DATA_BLOCK "T-84.00"   // DB53
VERSION : 0.1
// stored: AutoNumber false, DBAccessibleFromOPCUA true, DBAccessibleFromWebserver true, InstanceOfName Storage_Tank_Multi_Inload, InstanceOfType FB
"Storage_Tank_Multi_Inload"
BEGIN
END_DATA_BLOCK

DATA_BLOCK "T-85.00"   // DB52
VERSION : 0.1
// stored: AutoNumber false, DBAccessibleFromOPCUA true, DBAccessibleFromWebserver true, InstanceOfName Storage_Tank_Multi_Inload, InstanceOfType FB
"Storage_Tank_Multi_Inload"
BEGIN
END_DATA_BLOCK

DATA_BLOCK "T-02_ChiliAwetan_1"   // DB361
VERSION : 0.1
// stored: AutoNumber false, DBAccessibleFromOPCUA true, DBAccessibleFromWebserver true, InstanceOfName BFT_ChiliAwetan, InstanceOfType FB
"BFT_ChiliAwetan"
BEGIN
END_DATA_BLOCK

DATA_BLOCK "T-03_ChiliAwetan_2"   // DB362
VERSION : 0.1
// stored: AutoNumber false, DBAccessibleFromOPCUA true, DBAccessibleFromWebserver true, InstanceOfName BFT_ChiliAwetan, InstanceOfType FB
"BFT_ChiliAwetan"
BEGIN
END_DATA_BLOCK

DATA_BLOCK "T-04_ChiliAwetan_3"   // DB363
VERSION : 0.1
// stored: AutoNumber false, DBAccessibleFromOPCUA true, DBAccessibleFromWebserver true, InstanceOfName BFT_ChiliAwetan, InstanceOfType FB
"BFT_ChiliAwetan"
BEGIN
END_DATA_BLOCK

DATA_BLOCK "T-05_Tomato"   // DB364
VERSION : 0.1
// stored: AutoNumber false, DBAccessibleFromOPCUA true, DBAccessibleFromWebserver true, InstanceOfName BFT_Tomato, InstanceOfType FB
"BFT_Tomato"
BEGIN
END_DATA_BLOCK

DATA_BLOCK "T-06_ChiliFresh_1"   // DB365
VERSION : 0.1
// stored: AutoNumber false, DBAccessibleFromOPCUA true, DBAccessibleFromWebserver true, InstanceOfName BFT_ChiliFresh, InstanceOfType FB
"BFT_ChiliFresh"
BEGIN
END_DATA_BLOCK

DATA_BLOCK "T-07_ChiliFresh_2"   // DB366
VERSION : 0.1
// stored: AutoNumber false, DBAccessibleFromOPCUA true, DBAccessibleFromWebserver true, InstanceOfName BFT_ChiliFresh, InstanceOfType FB
"BFT_ChiliFresh"
BEGIN
END_DATA_BLOCK

DATA_BLOCK "T-08_ChiliFresh_3"   // DB367
VERSION : 0.1
// stored: AutoNumber false, DBAccessibleFromOPCUA true, DBAccessibleFromWebserver true, InstanceOfName BFT_ChiliFresh, InstanceOfType FB
"BFT_ChiliFresh"
BEGIN
END_DATA_BLOCK

DATA_BLOCK "T-09_Garlic"   // DB368
VERSION : 0.1
// stored: AutoNumber false, DBAccessibleFromOPCUA true, DBAccessibleFromWebserver true, InstanceOfName BFT_Garlic, InstanceOfType FB
"BFT_Garlic"
BEGIN
END_DATA_BLOCK

DATA_BLOCK "T-10_Vinegar"   // DB369
VERSION : 0.1
// stored: AutoNumber false, DBAccessibleFromOPCUA true, DBAccessibleFromWebserver true, InstanceOfName BFT_Vinegar, InstanceOfType FB
"BFT_Vinegar"
BEGIN
END_DATA_BLOCK

DATA_BLOCK "T-51_HW"   // DB370
VERSION : 0.1
// stored: AutoNumber false, DBAccessibleFromOPCUA true, DBAccessibleFromWebserver true, InstanceOfName Hot_Water, InstanceOfType FB
"Hot_Water"
BEGIN
END_DATA_BLOCK

DATA_BLOCK "BFT-61"   // DB111
VERSION : 0.1
// stored: AutoNumber false, DBAccessibleFromOPCUA true, DBAccessibleFromWebserver true, InstanceOfName Buffer_Tank, InstanceOfType FB
"Buffer_Tank"
BEGIN
END_DATA_BLOCK

DATA_BLOCK "BFT-64"   // DB112
VERSION : 0.1
// stored: AutoNumber false, DBAccessibleFromOPCUA true, DBAccessibleFromWebserver true, InstanceOfName Buffer_Tank, InstanceOfType FB
"Buffer_Tank"
BEGIN
END_DATA_BLOCK

DATA_BLOCK "BFT-65"   // DB113
VERSION : 0.1
// stored: AutoNumber false, DBAccessibleFromOPCUA true, DBAccessibleFromWebserver true, InstanceOfName Buffer_Tank, InstanceOfType FB
"Buffer_Tank"
BEGIN
END_DATA_BLOCK

DATA_BLOCK "BFT-66"   // DB114
VERSION : 0.1
// stored: AutoNumber false, DBAccessibleFromOPCUA true, DBAccessibleFromWebserver true, InstanceOfName Buffer_Tank, InstanceOfType FB
"Buffer_Tank"
BEGIN
END_DATA_BLOCK

DATA_BLOCK "BFT-67"   // DB115
VERSION : 0.1
// stored: AutoNumber false, DBAccessibleFromOPCUA true, DBAccessibleFromWebserver true, InstanceOfName Buffer_Tank, InstanceOfType FB
"Buffer_Tank"
BEGIN
END_DATA_BLOCK

DATA_BLOCK "BFT-68"   // DB116
VERSION : 0.1
// stored: AutoNumber false, DBAccessibleFromOPCUA true, DBAccessibleFromWebserver true, InstanceOfName Buffer_Tank, InstanceOfType FB
"Buffer_Tank"
BEGIN
END_DATA_BLOCK

DATA_BLOCK "Danfos_VSD_DB"   // DB46
VERSION : 0.1
// stored: AutoNumber false, DBAccessibleFromOPCUA true, DBAccessibleFromWebserver true, InstanceOfName Danfos_VSD, InstanceOfType FB
"Danfos_VSD"
BEGIN
END_DATA_BLOCK

DATA_BLOCK "IO Motor MCC Panel Blending_DB"   // DB5
VERSION : 0.1
// stored: AutoNumber true, DBAccessibleFromOPCUA true, DBAccessibleFromWebserver true, InstanceOfName IO Motor MCC Panel Blending, InstanceOfType FB
"IO Motor MCC Panel Blending"
BEGIN
   "XA-20.00".IN_SP_Speed := 5.0;
   "XA-21.00".IN_SP_Speed := 5.0;
   "P-21.01".IN_SP_Speed := 5.0;
   "XA-30.00".IN_SP_Speed := 5.0;
   "XA-31.00".IN_SP_Speed := 5.0;
   "P-31.01".IN_SP_Speed := 5.0;
   "P-32.01".IN_SP_Speed := 5.0;
   "P-32.03".IN_SP_Speed := 5.0;
END_DATA_BLOCK

DATA_BLOCK "P21.01Dan"   // DB23
VERSION : 0.1
// stored: AutoNumber true, DBAccessibleFromOPCUA true, DBAccessibleFromWebserver true, InstanceOfName Danfos_VSD, InstanceOfType FB
"Danfos_VSD"
BEGIN
END_DATA_BLOCK

DATA_BLOCK "P22.01Dan"   // DB22
VERSION : 0.1
// stored: AutoNumber true, DBAccessibleFromOPCUA true, DBAccessibleFromWebserver true, InstanceOfName Danfos_VSD, InstanceOfType FB
"Danfos_VSD"
BEGIN
END_DATA_BLOCK

DATA_BLOCK "IO Analog Homomixer_DB"   // DB2
VERSION : 0.1
// stored: AutoNumber true, DBAccessibleFromOPCUA true, DBAccessibleFromWebserver true, InstanceOfName IO Analog Homomixer, InstanceOfType FB
"IO Analog Homomixer"
BEGIN
END_DATA_BLOCK

DATA_BLOCK "IO Digital Homomixer_DB"   // DB3
VERSION : 0.1
// stored: AutoNumber true, DBAccessibleFromOPCUA true, DBAccessibleFromWebserver true, InstanceOfName IO Digital Homomixer, InstanceOfType FB
"IO Digital Homomixer"
BEGIN
END_DATA_BLOCK

DATA_BLOCK "IO Valve Homomixer_DB"   // DB4
VERSION : 0.1
// stored: AutoNumber true, DBAccessibleFromOPCUA true, DBAccessibleFromWebserver true, InstanceOfName IO Valve Homomixer, InstanceOfType FB
"IO Valve Homomixer"
BEGIN
END_DATA_BLOCK

DATA_BLOCK "IO Analog Blending_DB"   // DB6
VERSION : 0.1
// stored: AutoNumber true, DBAccessibleFromOPCUA true, DBAccessibleFromWebserver true, InstanceOfName IO Analog Blending, InstanceOfType FB
"IO Analog Blending"
BEGIN
END_DATA_BLOCK

DATA_BLOCK "IO Digital Blending_DB"   // DB7
VERSION : 0.1
// stored: AutoNumber true, DBAccessibleFromOPCUA true, DBAccessibleFromWebserver true, InstanceOfName IO Digital Blending, InstanceOfType FB
"IO Digital Blending"
BEGIN
END_DATA_BLOCK

DATA_BLOCK "IO_Valve_Blend20_DB"   // DB28
VERSION : 0.1
// stored: AutoNumber true, DBAccessibleFromOPCUA true, DBAccessibleFromWebserver true, InstanceOfName IO_Valve_Blend20, InstanceOfType FB
"IO_Valve_Blend20"
BEGIN
END_DATA_BLOCK

DATA_BLOCK "IO_Valve_Blend21_DB"   // DB39
VERSION : 0.1
// stored: AutoNumber true, DBAccessibleFromOPCUA true, DBAccessibleFromWebserver true, InstanceOfName IO_Valve_Blend21, InstanceOfType FB
"IO_Valve_Blend21"
BEGIN
END_DATA_BLOCK

DATA_BLOCK "IO_Valve_Blend30_DB"   // DB60
VERSION : 0.1
// stored: AutoNumber true, DBAccessibleFromOPCUA true, DBAccessibleFromWebserver true, InstanceOfName IO_Valve_Blend30, InstanceOfType FB
"IO_Valve_Blend30"
BEGIN
END_DATA_BLOCK

DATA_BLOCK "IO_Valve_Blend31_DB"   // DB61
VERSION : 0.1
// stored: AutoNumber true, DBAccessibleFromOPCUA true, DBAccessibleFromWebserver true, InstanceOfName IO_Valve_Blend31, InstanceOfType FB
"IO_Valve_Blend31"
BEGIN
END_DATA_BLOCK

DATA_BLOCK "IO_Valve_Blend40_DB"   // DB26
VERSION : 0.1
// stored: AutoNumber true, DBAccessibleFromOPCUA true, DBAccessibleFromWebserver true, InstanceOfName IO_Valve_Blend40, InstanceOfType FB
"IO_Valve_Blend40"
BEGIN
END_DATA_BLOCK

DATA_BLOCK "IO_Valve_Blend41_DB"   // DB62
VERSION : 0.1
// stored: AutoNumber true, DBAccessibleFromOPCUA true, DBAccessibleFromWebserver true, InstanceOfName IO_Valve_Blend41, InstanceOfType FB
"IO_Valve_Blend41"
BEGIN
END_DATA_BLOCK

DATA_BLOCK "IO_Valve_Blending_DB"   // DB8
VERSION : 0.1
// stored: AutoNumber true, DBAccessibleFromOPCUA true, DBAccessibleFromWebserver true, InstanceOfName IO_Valve_Blending, InstanceOfType FB
"IO_Valve_Blending"
BEGIN
   "AV-20.02".OPdwCmd := 16#0008_0000;
   "AV-20.03".OPdwCmd := 16#0008_0000;
   "AV-20.04".OPdwCmd := 16#0008_0000;
   "AV-20.05".OPdwCmd := 16#0008_0000;
   "AV-20.06".OPdwCmd := 16#0008_0000;
   "AV-20.07".OPdwCmd := 16#0008_0000;
   "AV-20.08".OPdwCmd := 16#0008_0000;
   "AV-20.09".OPdwCmd := 16#0008_0000;
   "AV-20.10".OPdwCmd := 16#0008_0000;
   "AV-20.11".OPdwCmd := 16#0008_0000;
   "AV-20.12".OPdwCmd := 16#0008_0000;
   "AV-20.13".OPdwCmd := 16#0008_0000;
   "AV-20.14".OPdwCmd := 16#0008_0000;
   "AV-20.15".OPdwCmd := 16#0008_0000;
   "AV-20.16".OPdwCmd := 16#0008_0000;
   "AV-20.17".OPdwCmd := 16#0008_0000;
   "AV-20.31".OPdwCmd := 16#0008_0000;
   "AV-20.32".OPdwCmd := 16#0008_0000;
   "AV-20.33".OPdwCmd := 16#0008_0000;
   "AV-20.34".OPdwCmd := 16#0008_0000;
   "AV-20.35".OPdwCmd := 16#0008_0000;
   "AV-20.36".OPdwCmd := 16#0008_0000;
   "AV-20.37".OPdwCmd := 16#0008_0000;
   "AV-20.38".OPdwCmd := 16#0008_0000;
   "AV-20.39".OPdwCmd := 16#0008_0000;
   "AV-20.40".OPdwCmd := 16#0008_0000;
   "AV-20.41".OPdwCmd := 16#0008_0000;
   "AV-21.01".OPdwCmd := 16#0008_0000;
   "AV-21.02".OPdwCmd := 16#0008_0000;
   "AV-21.03".OPdwCmd := 16#0008_0000;
   "AV-21.04".OPdwCmd := 16#0008_0000;
   "AV-21.05".OPdwCmd := 16#0008_0000;
   "AV-21.06".OPdwCmd := 16#0008_0000;
   "AV-21.07".OPdwCmd := 16#0008_0000;
   "AV-21.08".OPdwCmd := 16#0008_0000;
   "AV-21.09".OPdwCmd := 16#0008_0000;
   "AV-21.10".OPdwCmd := 16#0008_0000;
   "AV-21.11".OPdwCmd := 16#0008_0000;
   "AV-21.12".OPdwCmd := 16#0008_0000;
   "AV-21.13".OPdwCmd := 16#0008_0000;
   "AV-21.14".OPdwCmd := 16#0008_0000;
   "AV-21.15".OPdwCmd := 16#0008_0000;
   "AV-21.16".OPdwCmd := 16#0008_0000;
   "AV-21.17".OPdwCmd := 16#0008_0000;
   "AV-21.18".OPdwCmd := 16#0008_0000;
   "AV-21.31".OPdwCmd := 16#0008_0000;
   "AV-21.32".OPdwCmd := 16#0008_0000;
   "AV-21.33".OPdwCmd := 16#0008_0000;
   "AV-21.34".OPdwCmd := 16#0008_0000;
   "AV-21.35".OPdwCmd := 16#0008_0000;
   "AV-21.36".OPdwCmd := 16#0008_0000;
   "AV-21.37".OPdwCmd := 16#0008_0000;
   "AV-21.38".OPdwCmd := 16#0008_0000;
   "AV-21.39".OPdwCmd := 16#0008_0000;
   "AV-21.40".OPdwCmd := 16#0008_0000;
   "AV-21.41".OPdwCmd := 16#0008_0000;
   "AV-22.01".OPdwCmd := 16#0008_0000;
   "AV-22.02".OPdwCmd := 16#0008_0000;
   "AV-22.03".OPdwCmd := 16#0008_0000;
   "AV-22.06".OPdwCmd := 16#0008_0000;
   "AV-22.11".OPdwCmd := 16#0008_0000;
   "AV-22.21".OPdwCmd := 16#0008_0000;
   "AV-22.22".OPdwCmd := 16#0008_0000;
   "AV-30.01".OPdwCmd := 16#0008_0000;
   "AV-30.02".OPdwCmd := 16#0008_0000;
   "AV-30.03".OPdwCmd := 16#0008_0000;
   "AV-30.04".OPdwCmd := 16#0008_0000;
   "AV-30.05".OPdwCmd := 16#0008_0000;
   "AV-30.06".OPdwCmd := 16#0008_0000;
   "AV-30.07".OPdwCmd := 16#0008_0000;
   "AV-30.08".OPdwCmd := 16#0008_0000;
   "AV-30.09".OPdwCmd := 16#0008_0000;
   "AV-30.10".OPdwCmd := 16#0008_0000;
   "AV-30.11".OPdwCmd := 16#0008_0000;
   "AV-30.12".OPdwCmd := 16#0008_0000;
   "AV-30.13".OPdwCmd := 16#0008_0000;
   "AV-30.14".OPdwCmd := 16#0008_0000;
   "AV-30.15".OPdwCmd := 16#0008_0000;
   "AV-30.16".OPdwCmd := 16#0008_0000;
   "AV-30.17".OPdwCmd := 16#0008_0000;
   "AV-30.31".OPdwCmd := 16#0008_0000;
   "AV-30.32".OPdwCmd := 16#0008_0000;
   "AV-30.33".OPdwCmd := 16#0008_0000;
   "AV-30.34".OPdwCmd := 16#0008_0000;
   "AV-30.35".OPdwCmd := 16#0008_0000;
   "AV-30.36".OPdwCmd := 16#0008_0000;
   "AV-30.37".OPdwCmd := 16#0008_0000;
   "AV-30.38".OPdwCmd := 16#0008_0000;
   "AV-30.39".OPdwCmd := 16#0008_0000;
   "AV-30.40".OPdwCmd := 16#0008_0000;
   "AV-30.41".OPdwCmd := 16#0008_0000;
   "AV-31.01".OPdwCmd := 16#0008_0000;
   "AV-31.02".OPdwCmd := 16#0008_0000;
   "AV-31.03".OPdwCmd := 16#0008_0000;
   "AV-31.04".OPdwCmd := 16#0008_0000;
   "AV-31.05".OPdwCmd := 16#0008_0000;
   "AV-31.06".OPdwCmd := 16#0008_0000;
   "AV-31.07".OPdwCmd := 16#0008_0000;
   "AV-31.08".OPdwCmd := 16#0008_0000;
   "AV-31.09".OPdwCmd := 16#0008_0000;
   "AV-31.10".OPdwCmd := 16#0008_0000;
   "AV-31.11".OPdwCmd := 16#0008_0000;
   "AV-31.12".OPdwCmd := 16#0008_0000;
   "AV-31.13".OPdwCmd := 16#0008_0000;
   "AV-31.14".OPdwCmd := 16#0008_0000;
   "AV-31.15".OPdwCmd := 16#0008_0000;
   "AV-31.16".OPdwCmd := 16#0008_0000;
   "AV-31.17".OPdwCmd := 16#0008_0000;
   "AV-31.18".OPdwCmd := 16#0008_0000;
   "AV-31.31".OPdwCmd := 16#0008_0000;
   "AV-31.32".OPdwCmd := 16#0008_0000;
   "AV-31.33".OPdwCmd := 16#0008_0000;
   "AV-31.34".OPdwCmd := 16#0008_0000;
   "AV-31.35".OPdwCmd := 16#0008_0000;
   "AV-31.36".OPdwCmd := 16#0008_0000;
   "AV-31.37".OPdwCmd := 16#0008_0000;
   "AV-31.38".OPdwCmd := 16#0008_0000;
   "AV-31.39".OPdwCmd := 16#0008_0000;
   "AV-31.40".OPdwCmd := 16#0008_0000;
   "AV-31.41".OPdwCmd := 16#0008_0000;
   "AV-31.51".OPdwCmd := 16#0008_0000;
   "AV-31.52".OPdwCmd := 16#0008_0000;
   "AV-31.53".OPdwCmd := 16#0008_0000;
   "AV-31.54".OPdwCmd := 16#0008_0000;
   "AV-31.55".OPdwCmd := 16#0008_0000;
   "AV-31.56".OPdwCmd := 16#0008_0000;
   "AV-31.57".OPdwCmd := 16#0008_0000;
   "AV-31.58".OPdwCmd := 16#0008_0000;
   "AV-31.59".OPdwCmd := 16#0008_0000;
   "AV-31.60".OPdwCmd := 16#0008_0000;
   "AV-31.61".OPdwCmd := 16#0008_0000;
   "AV-31.62".OPdwCmd := 16#0008_0000;
   "AV-32.01".OPdwCmd := 16#0008_0000;
   "AV-32.02".OPdwCmd := 16#0008_0000;
   "AV-32.03".OPdwCmd := 16#0008_0000;
   "AV-32.06".OPdwCmd := 16#0008_0000;
   "AV-32.11".OPdwCmd := 16#0008_0000;
   "AV-32.21".OPdwCmd := 16#0008_0000;
   "AV-32.22".OPdwCmd := 16#0008_0000;
   "AV-20.42".OPdwCmd := 16#0008_0000;
   "AV-21.42".OPdwCmd := 16#0008_0000;
   "AV-22.04".OPdwCmd := 16#0008_0000;
   "AV-22.05".OPdwCmd := 16#0008_0000;
   "AV-30.42".OPdwCmd := 16#0008_0000;
   "AV-31.42".OPdwCmd := 16#0008_0000;
   "AV-32.04".OPdwCmd := 16#0008_0000;
   "AV-32.05".OPdwCmd := 16#0008_0000;
END_DATA_BLOCK

DATA_BLOCK "IO Analog Storage_DB"   // DB9
VERSION : 0.1
// stored: AutoNumber true, DBAccessibleFromOPCUA true, DBAccessibleFromWebserver true, InstanceOfName IO Analog Storage, InstanceOfType FB
"IO Analog Storage"
BEGIN
END_DATA_BLOCK

DATA_BLOCK "IO_Digital_Storage_DB"   // DB44
VERSION : 0.1
// stored: AutoNumber true, DBAccessibleFromOPCUA true, DBAccessibleFromWebserver true, InstanceOfName IO_Digital_Storage, InstanceOfType FB
"IO_Digital_Storage"
BEGIN
END_DATA_BLOCK

DATA_BLOCK "IO_Valve_Storage_DB"   // DB11
VERSION : 0.1
// stored: AutoNumber true, DBAccessibleFromOPCUA true, DBAccessibleFromWebserver true, InstanceOfName IO_Valve_Storage, InstanceOfType FB
"IO_Valve_Storage"
BEGIN
END_DATA_BLOCK

DATA_BLOCK "IO Motor MCC Preparation_DB"   // DB12
VERSION : 0.1
// stored: AutoNumber true, DBAccessibleFromOPCUA true, DBAccessibleFromWebserver true, InstanceOfName IO Motor MCC Preparation, InstanceOfType FB
"IO Motor MCC Preparation"
BEGIN
END_DATA_BLOCK

DATA_BLOCK "IO Analog Preparation_DB"   // DB13
VERSION : 0.1
// stored: AutoNumber true, DBAccessibleFromOPCUA true, DBAccessibleFromWebserver true, InstanceOfName IO Analog Preparation, InstanceOfType FB
"IO Analog Preparation"
BEGIN
END_DATA_BLOCK

DATA_BLOCK "IO Digital Preparation_DB"   // DB14
VERSION : 0.1
// stored: AutoNumber true, DBAccessibleFromOPCUA true, DBAccessibleFromWebserver true, InstanceOfName IO Digital Preparation, InstanceOfType FB
"IO Digital Preparation"
BEGIN
END_DATA_BLOCK

DATA_BLOCK "IO_Valve_T01_HWT"   // DB301
VERSION : 0.1
// stored: AutoNumber false, DBAccessibleFromOPCUA true, DBAccessibleFromWebserver true, InstanceOfName IO Valve T01 HWT, InstanceOfType FB
"IO Valve T01 HWT"
BEGIN
END_DATA_BLOCK

DATA_BLOCK "IO_Valve_T02_Chili"   // DB302
VERSION : 0.1
// stored: AutoNumber false, DBAccessibleFromOPCUA true, DBAccessibleFromWebserver true, InstanceOfName IO Valve T02 Chili, InstanceOfType FB
"IO Valve T02 Chili"
BEGIN
END_DATA_BLOCK

DATA_BLOCK "IO_Valve_T03_Chili"   // DB303
VERSION : 0.1
// stored: AutoNumber false, DBAccessibleFromOPCUA true, DBAccessibleFromWebserver true, InstanceOfName IO Valve T03 Chili, InstanceOfType FB
"IO Valve T03 Chili"
BEGIN
END_DATA_BLOCK

DATA_BLOCK "IO_Valve_T04_Chili"   // DB304
VERSION : 0.1
// stored: AutoNumber false, DBAccessibleFromOPCUA true, DBAccessibleFromWebserver true, InstanceOfName IO Valve T04 Chili, InstanceOfType FB
"IO Valve T04 Chili"
BEGIN
END_DATA_BLOCK

DATA_BLOCK "IO_Valve_T05_Tomato"   // DB305
VERSION : 0.1
// stored: AutoNumber false, DBAccessibleFromOPCUA true, DBAccessibleFromWebserver true, InstanceOfName IO Valve T05 Tomato, InstanceOfType FB
"IO Valve T05 Tomato"
BEGIN
END_DATA_BLOCK

DATA_BLOCK "IO_Valve_T06_FreshChili"   // DB306
VERSION : 0.1
// stored: AutoNumber false, DBAccessibleFromOPCUA true, DBAccessibleFromWebserver true, InstanceOfName IO Valve T06 FreshChili, InstanceOfType FB
"IO Valve T06 FreshChili"
BEGIN
END_DATA_BLOCK

DATA_BLOCK "IO_Valve_T07_FreshChili"   // DB307
VERSION : 0.1
// stored: AutoNumber false, DBAccessibleFromOPCUA true, DBAccessibleFromWebserver true, InstanceOfName IO Valve T07 FreshChili, InstanceOfType FB
"IO Valve T07 FreshChili"
BEGIN
END_DATA_BLOCK

DATA_BLOCK "IO_Valve_T08_FreshChili"   // DB308
VERSION : 0.1
// stored: AutoNumber false, DBAccessibleFromOPCUA true, DBAccessibleFromWebserver true, InstanceOfName IO Valve T08 FreshChili, InstanceOfType FB
"IO Valve T08 FreshChili"
BEGIN
END_DATA_BLOCK

DATA_BLOCK "IO_Valve_T09_Garlic"   // DB309
VERSION : 0.1
// stored: AutoNumber false, DBAccessibleFromOPCUA true, DBAccessibleFromWebserver true, InstanceOfName IO Valve T09 Garlic, InstanceOfType FB
"IO Valve T09 Garlic"
BEGIN
END_DATA_BLOCK

DATA_BLOCK "IO_Valve_T10_Vinegar"   // DB310
VERSION : 0.1
// stored: AutoNumber false, DBAccessibleFromOPCUA true, DBAccessibleFromWebserver true, InstanceOfName IO Valve T10 Vinegar, InstanceOfType FB
"IO Valve T10 Vinegar"
BEGIN
END_DATA_BLOCK

DATA_BLOCK "IO_Valve_T51_HW"   // DB311
VERSION : 0.1
// stored: AutoNumber false, DBAccessibleFromOPCUA true, DBAccessibleFromWebserver true, InstanceOfName IO Valve T51 HotWaterLine, InstanceOfType FB
"IO Valve T51 HotWaterLine"
BEGIN
END_DATA_BLOCK

DATA_BLOCK "IO_Valve_Buffer_DB"   // DB64
VERSION : 0.1
// stored: AutoNumber true, DBAccessibleFromOPCUA true, DBAccessibleFromWebserver true, InstanceOfName IO_Valve_Buffer, InstanceOfType FB
"IO_Valve_Buffer"
BEGIN
END_DATA_BLOCK

DATA_BLOCK "Totalizer_FT-00.01"   // DB381
VERSION : 0.1
// stored: AutoNumber false, DBAccessibleFromOPCUA true, DBAccessibleFromWebserver true, InstanceOfName Totalizer, InstanceOfType FB
"Totalizer"
BEGIN
END_DATA_BLOCK

DATA_BLOCK "Totalizer_FT-02.01"   // DB382
VERSION : 0.1
// stored: AutoNumber false, DBAccessibleFromOPCUA true, DBAccessibleFromWebserver true, InstanceOfName Totalizer, InstanceOfType FB
"Totalizer"
BEGIN
END_DATA_BLOCK

DATA_BLOCK "Totalizer_FT-03.01"   // DB383
VERSION : 0.1
// stored: AutoNumber false, DBAccessibleFromOPCUA true, DBAccessibleFromWebserver true, InstanceOfName Totalizer, InstanceOfType FB
"Totalizer"
BEGIN
END_DATA_BLOCK

DATA_BLOCK "Totalizer_FT-04.01"   // DB384
VERSION : 0.1
// stored: AutoNumber false, DBAccessibleFromOPCUA true, DBAccessibleFromWebserver true, InstanceOfName Totalizer, InstanceOfType FB
"Totalizer"
BEGIN
END_DATA_BLOCK

DATA_BLOCK "Totalizer_FT-05.01"   // DB385
VERSION : 0.1
// stored: AutoNumber false, DBAccessibleFromOPCUA true, DBAccessibleFromWebserver true, InstanceOfName Totalizer, InstanceOfType FB
"Totalizer"
BEGIN
END_DATA_BLOCK

DATA_BLOCK "Totalizer_FT-06.01"   // DB386
VERSION : 0.1
// stored: AutoNumber false, DBAccessibleFromOPCUA true, DBAccessibleFromWebserver true, InstanceOfName Totalizer, InstanceOfType FB
"Totalizer"
BEGIN
END_DATA_BLOCK

DATA_BLOCK "Totalizer_FT-07.01"   // DB387
VERSION : 0.1
// stored: AutoNumber false, DBAccessibleFromOPCUA true, DBAccessibleFromWebserver true, InstanceOfName Totalizer, InstanceOfType FB
"Totalizer"
BEGIN
END_DATA_BLOCK

DATA_BLOCK "Totalizer_FT-08.01"   // DB388
VERSION : 0.1
// stored: AutoNumber false, DBAccessibleFromOPCUA true, DBAccessibleFromWebserver true, InstanceOfName Totalizer, InstanceOfType FB
"Totalizer"
BEGIN
END_DATA_BLOCK

DATA_BLOCK "Totalizer_FT-09.01"   // DB389
VERSION : 0.1
// stored: AutoNumber false, DBAccessibleFromOPCUA true, DBAccessibleFromWebserver true, InstanceOfName Totalizer, InstanceOfType FB
"Totalizer"
BEGIN
END_DATA_BLOCK

DATA_BLOCK "Totalizer_FT-10.01"   // DB390
VERSION : 0.1
// stored: AutoNumber false, DBAccessibleFromOPCUA true, DBAccessibleFromWebserver true, InstanceOfName Totalizer, InstanceOfType FB
"Totalizer"
BEGIN
END_DATA_BLOCK

DATA_BLOCK "Totalizer_FT-12.01"   // DB393
VERSION : 0.1
// stored: AutoNumber false, DBAccessibleFromOPCUA true, DBAccessibleFromWebserver true, InstanceOfName Totalizer, InstanceOfType FB
"Totalizer"
BEGIN
END_DATA_BLOCK

DATA_BLOCK "Totalizer_FT-12.02"   // DB394
VERSION : 0.1
// stored: AutoNumber false, DBAccessibleFromOPCUA true, DBAccessibleFromWebserver true, InstanceOfName Totalizer, InstanceOfType FB
"Totalizer"
BEGIN
END_DATA_BLOCK

DATA_BLOCK "Totalizer_FT-51.01"   // DB391
VERSION : 0.1
// stored: AutoNumber false, DBAccessibleFromOPCUA true, DBAccessibleFromWebserver true, InstanceOfName Totalizer, InstanceOfType FB
"Totalizer"
BEGIN
END_DATA_BLOCK

DATA_BLOCK "GET_DB_1"   // DB27
// stored: AutoNumber true, DBAccessibleFromOPCUA true, DBAccessibleFromWebserver true, InstanceOfName GET_SFB, OfSystemLibElement GET, OfSystemLibVersion 1.2
"GET_SFB"
   // VAR_INPUT
   //    REQ : Bool;
   //    ID : Word;
   // END_VAR
   // VAR_OUTPUT
   //    NDR : Bool;
   //    ERROR : Bool;
   //    STATUS : Word;
   // END_VAR
   // VAR_IN_OUT
   //    ADDR_1 : Remote;
   //    ADDR_2 : Remote;
   //    ADDR_3 : Remote;
   //    ADDR_4 : Remote;
   //    RD_1 : Variant;
   //    RD_2 : Variant;
   //    RD_3 : Variant;
   //    RD_4 : Variant;
   // END_VAR
BEGIN
END_DATA_BLOCK

DATA_BLOCK "GET_OSA_CIP"   // DB50
// stored: AutoNumber false, DBAccessibleFromOPCUA true, DBAccessibleFromWebserver true, InstanceOfName GET_SFB, OfSystemLibElement GET, OfSystemLibVersion 1.2
"GET_SFB"
   // VAR_INPUT
   //    REQ : Bool;
   //    ID : Word;
   // END_VAR
   // VAR_OUTPUT
   //    NDR : Bool;
   //    ERROR : Bool;
   //    STATUS : Word;
   // END_VAR
   // VAR_IN_OUT
   //    ADDR_1 : Remote;
   //    ADDR_2 : Remote;
   //    ADDR_3 : Remote;
   //    ADDR_4 : Remote;
   //    RD_1 : Variant;
   //    RD_2 : Variant;
   //    RD_3 : Variant;
   //    RD_4 : Variant;
   // END_VAR
BEGIN
END_DATA_BLOCK

DATA_BLOCK "GET_OSA_Chili"   // DB57
// stored: AutoNumber false, DBAccessibleFromOPCUA true, DBAccessibleFromWebserver true, InstanceOfName GET_SFB, OfSystemLibElement GET, OfSystemLibVersion 1.2
"GET_SFB"
   // VAR_INPUT
   //    REQ : Bool;
   //    ID : Word;
   // END_VAR
   // VAR_OUTPUT
   //    NDR : Bool;
   //    ERROR : Bool;
   //    STATUS : Word;
   // END_VAR
   // VAR_IN_OUT
   //    ADDR_1 : Remote;
   //    ADDR_2 : Remote;
   //    ADDR_3 : Remote;
   //    ADDR_4 : Remote;
   //    RD_1 : Variant;
   //    RD_2 : Variant;
   //    RD_3 : Variant;
   //    RD_4 : Variant;
   // END_VAR
BEGIN
END_DATA_BLOCK

DATA_BLOCK "Get_Tipper1"   // DB242
// stored: AutoNumber false, DBAccessibleFromOPCUA true, DBAccessibleFromWebserver true, InstanceOfName GET_SFB, OfSystemLibElement GET, OfSystemLibVersion 1.2
"GET_SFB"
   // VAR_INPUT
   //    REQ : Bool;
   //    ID : Word;
   // END_VAR
   // VAR_OUTPUT
   //    NDR : Bool;
   //    ERROR : Bool;
   //    STATUS : Word;
   // END_VAR
   // VAR_IN_OUT
   //    ADDR_1 : Remote;
   //    ADDR_2 : Remote;
   //    ADDR_3 : Remote;
   //    ADDR_4 : Remote;
   //    RD_1 : Variant;
   //    RD_2 : Variant;
   //    RD_3 : Variant;
   //    RD_4 : Variant;
   // END_VAR
BEGIN
END_DATA_BLOCK

DATA_BLOCK "Get_Tipper2"   // DB246
// stored: AutoNumber false, DBAccessibleFromOPCUA true, DBAccessibleFromWebserver true, InstanceOfName GET_SFB, OfSystemLibElement GET, OfSystemLibVersion 1.2
"GET_SFB"
   // VAR_INPUT
   //    REQ : Bool;
   //    ID : Word;
   // END_VAR
   // VAR_OUTPUT
   //    NDR : Bool;
   //    ERROR : Bool;
   //    STATUS : Word;
   // END_VAR
   // VAR_IN_OUT
   //    ADDR_1 : Remote;
   //    ADDR_2 : Remote;
   //    ADDR_3 : Remote;
   //    ADDR_4 : Remote;
   //    RD_1 : Variant;
   //    RD_2 : Variant;
   //    RD_3 : Variant;
   //    RD_4 : Variant;
   // END_VAR
BEGIN
END_DATA_BLOCK

DATA_BLOCK "PUT_OSA_CIP"   // DB56
// stored: AutoNumber false, DBAccessibleFromOPCUA true, DBAccessibleFromWebserver true, InstanceOfName PUT_SFB, OfSystemLibElement PUT, OfSystemLibVersion 1.3
"PUT_SFB"
   // VAR_INPUT
   //    REQ : Bool;
   //    ID : Word;
   // END_VAR
   // VAR_OUTPUT
   //    DONE : Bool;
   //    ERROR : Bool;
   //    STATUS : Word;
   // END_VAR
   // VAR_IN_OUT
   //    ADDR_1 : Remote;
   //    ADDR_2 : Remote;
   //    ADDR_3 : Remote;
   //    ADDR_4 : Remote;
   //    SD_1 : Variant;
   //    SD_2 : Variant;
   //    SD_3 : Variant;
   //    SD_4 : Variant;
   // END_VAR
BEGIN
END_DATA_BLOCK

DATA_BLOCK "PUT_OSA_Chili"   // DB58
// stored: AutoNumber true, DBAccessibleFromOPCUA true, DBAccessibleFromWebserver true, InstanceOfName PUT_SFB, OfSystemLibElement PUT, OfSystemLibVersion 1.3
"PUT_SFB"
   // VAR_INPUT
   //    REQ : Bool;
   //    ID : Word;
   // END_VAR
   // VAR_OUTPUT
   //    DONE : Bool;
   //    ERROR : Bool;
   //    STATUS : Word;
   // END_VAR
   // VAR_IN_OUT
   //    ADDR_1 : Remote;
   //    ADDR_2 : Remote;
   //    ADDR_3 : Remote;
   //    ADDR_4 : Remote;
   //    SD_1 : Variant;
   //    SD_2 : Variant;
   //    SD_3 : Variant;
   //    SD_4 : Variant;
   // END_VAR
BEGIN
END_DATA_BLOCK

DATA_BLOCK "Put_Tipper1"   // DB243
// stored: AutoNumber false, DBAccessibleFromOPCUA true, DBAccessibleFromWebserver true, InstanceOfName PUT_SFB, OfSystemLibElement PUT, OfSystemLibVersion 1.3
"PUT_SFB"
   // VAR_INPUT
   //    REQ : Bool;
   //    ID : Word;
   // END_VAR
   // VAR_OUTPUT
   //    DONE : Bool;
   //    ERROR : Bool;
   //    STATUS : Word;
   // END_VAR
   // VAR_IN_OUT
   //    ADDR_1 : Remote;
   //    ADDR_2 : Remote;
   //    ADDR_3 : Remote;
   //    ADDR_4 : Remote;
   //    SD_1 : Variant;
   //    SD_2 : Variant;
   //    SD_3 : Variant;
   //    SD_4 : Variant;
   // END_VAR
BEGIN
END_DATA_BLOCK

DATA_BLOCK "Put_Tipper2"   // DB247
// stored: AutoNumber false, DBAccessibleFromOPCUA true, DBAccessibleFromWebserver true, InstanceOfName PUT_SFB, OfSystemLibElement PUT, OfSystemLibVersion 1.3
"PUT_SFB"
   // VAR_INPUT
   //    REQ : Bool;
   //    ID : Word;
   // END_VAR
   // VAR_OUTPUT
   //    DONE : Bool;
   //    ERROR : Bool;
   //    STATUS : Word;
   // END_VAR
   // VAR_IN_OUT
   //    ADDR_1 : Remote;
   //    ADDR_2 : Remote;
   //    ADDR_3 : Remote;
   //    ADDR_4 : Remote;
   //    SD_1 : Variant;
   //    SD_2 : Variant;
   //    SD_3 : Variant;
   //    SD_4 : Variant;
   // END_VAR
BEGIN
END_DATA_BLOCK

DATA_BLOCK "Timer_Pulse_Drain_Water_THE1"   // DB30
{ S7_Optimized_Access := 'TRUE' }
// stored: AutoNumber true, DBAccessibleFromOPCUA true, DBAccessibleFromWebserver true, InstanceOfName IEC_TIMER, OfSystemLibElement IEC_TIMER, OfSystemLibVersion 1.0
"IEC_TIMER"
   // VAR
   //    PT : Time := T#15s;
   //    ET { ExternalWritable := 'False'} : Time;
   //    IN : Bool;
   //    Q { ExternalWritable := 'False'} : Bool;
   // END_VAR
BEGIN
END_DATA_BLOCK

DATA_BLOCK "Timer_Pulse_Drain_Water_THE2"   // DB29
{ S7_Optimized_Access := 'TRUE' }
// stored: AutoNumber true, DBAccessibleFromOPCUA true, DBAccessibleFromWebserver true, InstanceOfName IEC_TIMER, OfSystemLibElement IEC_TIMER, OfSystemLibVersion 1.0
"IEC_TIMER"
   // VAR
   //    PT : Time := T#15s;
   //    ET { ExternalWritable := 'False'} : Time;
   //    IN : Bool;
   //    Q { ExternalWritable := 'False'} : Bool;
   // END_VAR
BEGIN
END_DATA_BLOCK

DATA_BLOCK "Rework_T-22_DB"   // DB48
VERSION : 0.1
// stored: AutoNumber false, DBAccessibleFromOPCUA true, DBAccessibleFromWebserver true, InstanceOfName Rework, InstanceOfType FB
"Rework"
BEGIN
END_DATA_BLOCK

DATA_BLOCK "Rework_T-32_DB"   // DB49
VERSION : 0.1
// stored: AutoNumber false, DBAccessibleFromOPCUA true, DBAccessibleFromWebserver true, InstanceOfName Rework, InstanceOfType FB
"Rework"
BEGIN
END_DATA_BLOCK

DATA_BLOCK "T-20.00_DB"   // DB18
VERSION : 0.1
// stored: AutoNumber true, DBAccessibleFromOPCUA true, DBAccessibleFromWebserver true, InstanceOfName BLEND, InstanceOfType FB
"BLEND"
BEGIN
END_DATA_BLOCK

DATA_BLOCK "T-21.00_DB"   // DB19
VERSION : 0.1
// stored: AutoNumber true, DBAccessibleFromOPCUA true, DBAccessibleFromWebserver true, InstanceOfName BLEND, InstanceOfType FB
"BLEND"
BEGIN
END_DATA_BLOCK

DATA_BLOCK "T-30.00_DB"   // DB24
VERSION : 0.1
// stored: AutoNumber true, DBAccessibleFromOPCUA true, DBAccessibleFromWebserver true, InstanceOfName BLEND, InstanceOfType FB
"BLEND"
BEGIN
END_DATA_BLOCK

DATA_BLOCK "T-31.00_DB"   // DB25
VERSION : 0.1
// stored: AutoNumber true, DBAccessibleFromOPCUA true, DBAccessibleFromWebserver true, InstanceOfName BLEND, InstanceOfType FB
"BLEND"
BEGIN
END_DATA_BLOCK

DATA_BLOCK "T-01.01_DB"   // DB351
VERSION : 0.1
// stored: AutoNumber false, DBAccessibleFromOPCUA true, DBAccessibleFromWebserver true, InstanceOfName HWT, InstanceOfType FB
"HWT"
   // VAR_INPUT
   //    "IN_FBAV.01" : Bool;
   //    "IN_FBAV.02" : Bool;
   //    "IN_FBAV.03" : Bool;
   //    "IN_FBAV.04" : Bool;
   //    "IN_FBAV.10" : Bool;
   //    "IN_FBCV.10" : Bool;
   //    "IN_FS.01" : Bool;
   //    IN_LT01 : Real;
   //    IN_TT01 : Real;
   //    IN_TT02 : Real;
   //    "IN_FBP.01" : Bool;
   //    "IN_P.01-Speed" : Real;
   //    DosePumpSpeed : Real;
   //    "DoseON-OFF" : Bool;
   //    "DosePumpON-OFF" : Bool;
   //    CIPPulse : Bool;
   //    Line_OK : Bool;
   // END_VAR
   // VAR_OUTPUT
   //    "OUT_AV.01" : Bool;
   //    "OUT_AV.02" : Bool;
   //    "OUT_AV.03" : Bool;
   //    "OUT_AV.04" : Bool;
   //    "OUT_AV.10" : Bool;
   //    "OUT_CV.10" : Bool;
   //    Q_PID_Setpoint : Real;
   //    Q_PID_PV_IN : Real;
   //    "OUT_FS.01" : Bool;
   //    "OUT_LT.01" : Real;
   //    "OUT_TT.01" : Real;
   //    "OUT_TT.02" : Real;
   //    "OUT_P.01" : Bool;
   //    "OUT_P.01-Speed" : Real;
   //    OUT_CIP_Request : Bool;
   //    Q_WH_Tank_Ready : Bool;
   // END_VAR
   // VAR
   //    Cmd : Struct
   //       Start_Prosses : Bool;
   //       Start_Preheat : Bool;
   //       HWT_Mode : Bool;
   //       Ready_for_Mix : Bool;
   //       "CIP Request" : Bool;
   //       Pump_Mode : Bool;
   //       Pump_Man_ON_OFF : Bool;
   //    END_STRUCT;
   //    Param : Struct
   //       SP_Level_LL : Real;
   //       SP_Level_ML : Real;
   //       SP_Level_HL : Real;
   //       SP_Temp_Prepar : Real;
   //       SP_Temp_Process : Real;
   //       SP_PumpSpeed : Real;
   //       L_Hi_Lim : Real;
   //       L_Lo_Lim : Real;
   //       L_Hys : Real;
   //       T_Hi_Lim : Real;
   //       T_Lo_Lim : Real;
   //       T_Hys : Real;
   //       CIP_Ret_ON_SP : Real;
   //       CIP_Ret_OFF_SP : Real;
   //    END_STRUCT;
   //    State : Struct
   //       Tank_LL : Bool;
   //       Tank_ML : Bool;
   //       Tank_HL : Bool;
   //       Temp_Preheat_OK : Bool;
   //       Temp_Process_OK : Bool;
   //       Tank_Heating : Bool;
   //       "Tank is Ready" : Bool;
   //       "Tank in transfer" : Bool;
   //       Enable_WHT_Mode : Bool;
   //       Enable_Ready : Bool;
   //       Ready_for_Mix : Bool;
   //       "CIP Request Enable" : Bool;
   //       "Tank in CIP" : Bool;
   //       CIP_Request_OK : Bool;
   //       CIP_ReturnON : Bool;
   //       HWT_Status : Int;
   //       Temp_Actual : Real;
   //    END_STRUCT;
   //    L_Hys_Abs : Real;
   //    T_Hys_Abs : Real;
   //    Hys_Level_HL : Real;
   //    Hys_Level_ML : Real;
   //    Hys_Level_LL : Real;
   //    "Hys SP_SP_Prepar" : Real;
   //    "Hys SP_SP_Process" : Real;
   //    "Hys SP_SP_" : Real;
   //    alwaysON : Bool;
   //    r : Struct
   //       PosE1 : Bool;
   //       PosE2 : Bool;
   //       PosE3 : Bool;
   //       PosE4 : Bool;
   //       PosE5 : Bool;
   //       PosE6 : Bool;
   //       PosE7 : Bool;
   //       PosE8 : Bool;
   //       PosE9 : Bool;
   //       PosE10 : Bool;
   //       PosE11 : Bool;
   //       PosE12 : Bool;
   //       PosE13 : Bool;
   //       PosE14 : Bool;
   //       PosE15 : Bool;
   //       PosE16 : Bool;
   //       PosE17 : Bool;
   //       PosE18 : Bool;
   //       PosE19 : Bool;
   //       PosE20 : Bool;
   //       PosE21 : Bool;
   //       PosE22 : Bool;
   //       PosE23 : Bool;
   //       PosE24 : Bool;
   //       PosE25 : Bool;
   //       PosE26 : Bool;
   //       PosE27 : Bool;
   //       PosE28 : Bool;
   //       PosE29 : Bool;
   //       PosE30 : Bool;
   //       PosE31 : Bool;
   //       PosE32 : Bool;
   //    END_STRUCT;
   //    Actuator : Struct
   //       AV_Inlet : Bool;
   //       AV_Return : Bool;
   //       CV_Steam : Bool;
   //       Pump : Bool;
   //    END_STRUCT;
   //    r_Pump : Bool;
   //    r_PumpTim { S7_SetPoint := 'True'} : IEC_TIMER;
   //    Alarm : Word;
   //    Event : Word;
   // END_VAR
BEGIN
END_DATA_BLOCK
